# EPICS StreamDevice protocol: agilent33220AApp/protocol/agilent33220A.proto
# 	streamDevice protocol file for Agilent Model 33210A Arbitrary Waveform Generator
# Based on ag33210a from triumf

InTerminator = '\n';
OutTerminator = '\n';
# MaxInput = 0;
# LockTimeout should be GT ReplyTimeout
LockTimeout = 2000;
ReplyTimeout = 300;
ReadTimeout = 100;

read_float {
    out "\$1?"; in "%f";
}

write_float {
    out "\$1 %e";
    @init{ read_float; }
}

read_int {
    out "\$1?"; in "%d";
}

write_int {
    out "\$1 %d";
    @init{ read_int;}
}

read_string {
    out "\$1?"; in "%s";
}

write_string {
    out "\$1 %s";
    @init{ read_string;}
}
